Fanuc KAREL source: kd00074.KL

-- PROVISIONAL review KL for V940-1; original PC SHA256 c6c1e4c17ef54c6071e5fa181728565a8af310a901b97360b768d113eac1e7cc
-- Incomplete behavior may be omitted. Consult companion uncertainty JSON. Do not deploy.
PROGRAM KD00074
%NOLOCKGROUP
VAR
  I : INTEGER
  J : INTEGER
  B : BOOLEAN
  R : REAL
  S : STRING[80]
BEGIN
  -- V9_ZERO_TABLE_METADATA_HINT layout=0001; no indexed target words; source/name/runtime held
  -- UNRESOLVED_PC offsets 5-7; opcodes 9C,3B
  -- UNRESOLVED_PC offsets 12-16; opcodes 7F
END KD00074
